{attribute 'GeneratedUsingTerminal: IODEVICETYPE_ETHERCATPROT'}
{attribute addProperty BoxType "IODEVICETYPE_ETHERCATPROT"}
{attribute addProperty Id "TcTerminals210_2EK1100TcTerminals210_2EK1100_50C143310SyncUnitsSyncUnits_99E584AF18InputsInputs_25A0042B160OutputsOutputs_2397A10E106InfoDataInfoData_E68C61CD28"}
{attribute addProperty CRC "2975250814"}
{attribute addProperty Size "312"}
{attribute addProperty Name "EtherCAT Master KL"}
TYPE EtherCAT_Master_KL_B156B97E EXTENDS EtcMasterBase_62654B43 :
STRUCT
	{attribute addProperty Name "TcTerminals210_2EK1100"}
	{attribute addProperty PreviousPort "EtherCAT Master KL : Master"}
	TcTerminals210_2EK1100 : TcTerminals210_2EK1100_50C14331;
	{attribute addProperty Name "SyncUnits"}
	SyncUnits : SyncUnits_99E584AF;
	{attribute addProperty Name "Inputs"}
	Inputs : Inputs_25A0042B;
	{attribute addProperty Name "Outputs"}
	Outputs : Outputs_2397A10E;
	{attribute addProperty Name "InfoData"}
	InfoData : InfoData_E68C61CD;
END_STRUCT
END_TYPE

(* stored: Version 1.2.0.0, ProductVersion 3.1.4024.11
   DUT EtherCAT_Master_KL_B156B97E: Id {91f15081-5aa9-494c-8079-0cc5a525bd30} *)
